(* PLC project Tc2_Utilities.UTF8Len Demo, tc3-libraries-kb TwinCAT 3.1 *)
(* stored: creationDateTime 2026-05-10T16:00:00, modificationDateTime 2026-05-10T16:00:00 *)

PROGRAM P_Demo_UTF8Len
  VAR
    rResult : UDINT;  (* UTF8Len 返回值 *)
    bRun : BOOL;  (* 触发一次调用 *)
    sUtf8 : STRING;  (* 测试用本地变量 *)
    bAsc : BOOL;  (* 测试用本地变量 *)
    nSz : UDINT;  (* 测试用本地变量 *)
  END_VAR

            // ============================================================
// Tc2_Utilities.UTF8Len 演示程序（FUNCTION）
// ============================================================
// 验证步骤：
//   1. 引用 Tc2_Utilities
//   2. 编译 + 登录
//   3. 强制 bRun := TRUE 一个周期
//   4. 在线监视 rResult / 各 demo 变量
// ============================================================

sUtf8 := sLiteral_TO_UTF8('café');
IF bRun THEN
    rResult := UTF8Len(pUTF8 := ADR(sUtf8), bASCII => bAsc, nSize => nSz);
    bRun := FALSE;
END_IF;

          
END_PROGRAM
